// TIA Portal V18 export
FUNCTION_BLOCK "Motor control function FB"   // FB1, LAD
{ S7_Optimized_Access := 'TRUE' }
VERSION : 0.1
// stored: AutoNumber true, IsIECCheckEnabled false, IsRetainMemResEnabled false, MemoryReserve 100, SetENOAutomatically false, UDAEnableTagReadback false
   VAR_INPUT
      "FB Start" : Bool;
      "FB Stop" : Bool;
      "FB CB Feedback" : Bool;
   END_VAR
   VAR_OUTPUT
      "FB Motor contactor" : Bool;
   END_VAR
BEGIN

REGION Network 1: Start motor contactor
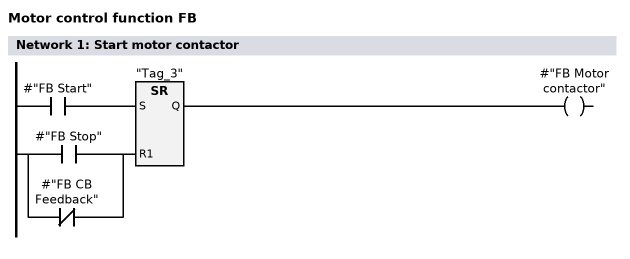
   RUNG wire#powerrail
      Contact( #"FB Start" )
      S_SR(operand := "Tag_3", r1 := wire#w1)
      Coil( #"FB Motor contactor" )
   END_RUNG
   RUNG wire#powerrail
      Contact( #"FB Stop" )
   END_RUNG wire#w1
   RUNG wire#powerrail
      I_Contact( #"FB CB Feedback" )
   END_RUNG wire#w1
   // the same network as SCL:
   IF #"FB Start" THEN
       "Tag_3" := TRUE;   // SR flip-flop
   END_IF;
   IF #"FB Stop" OR NOT #"FB CB Feedback" THEN "Tag_3" := FALSE; END_IF;
   #"FB Motor contactor" := "Tag_3";
END_REGION
END_FUNCTION_BLOCK
